TYPE ST_MachineStatus :
STRUCT
	////////////////////////////:
	eMachineState				:E_MachineState;
	
	// Status Flags:
	bSystemPowerUp 				:BOOL;
	bStopped 					:BOOL;
	bInitialising 				:BOOL;
	bReadyToStart 				:BOOL;
	bAutoCycle 					:BOOL;
	bStopping					:BOOL;
	bFault 						:BOOL;
	bManualMode					:BOOL;
	bSafety						:BOOL;

END_STRUCT
END_TYPE

(* stored: Version 1.1.0.1, ProductVersion 3.1.4026.17
   DUT ST_MachineStatus: Id {2fcb39d9-b828-4718-8c76-1a935a816f27} *)
